// Mitsubishi GX Works2 project: multi_prog   PLC: Q02/Q02H

PROGRAM part_1
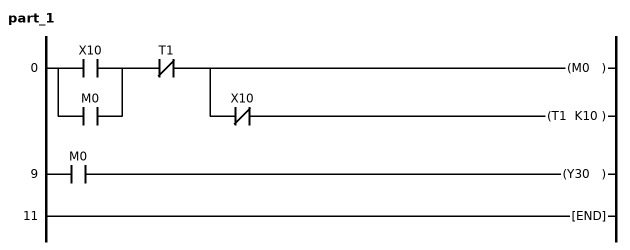
0     LD      X10
      OR      M0
      ANI     T1
      OUT     M0
      ANI     X10
      OUT     T1 K10
9     LD      M0
      OUT     Y30
11    END
END_PROGRAM

PROGRAM part_2
0     END
END_PROGRAM
